// Valid on Done (S3.10).
TYPE ST_RobotOutCmd :
STRUCT
    ReachedId : DWORD;   // position actually reached
END_STRUCT
END_TYPE

(* stored: Version 1.1.0.1, ProductVersion 3.1.4024.12
   DUT ST_RobotOutCmd: Id {3e53d771-8aac-433c-8244-806ed67cc6c9} *)
